Fanuc KAREL source: kb00161.KL

-- PROVISIONAL review KL for V940-1; original PC SHA256 606e9ad75cf5cc1266365447fe72f35daecf91610dc58aa2e1af25bdaba1c935
-- Incomplete behavior may be omitted. Consult companion uncertainty JSON. Do not deploy.
PROGRAM KB00161
%NOLOCKGROUP
BEGIN
  -- V9_ZERO_TABLE_METADATA_HINT layout=0002_ascii; no indexed target words; source/name/runtime held
  -- UNRESOLVED_PC offsets 5-12; opcodes 9D,23
  -- UNRESOLVED_PC offsets 17-24; opcodes 9D,23
  -- UNRESOLVED_PC offsets 29-59; opcodes 27,22,22,1C,22,27,9D,31
  -- UNRESOLVED_PC offsets 64-68; opcodes 7F
END KB00161
